Yaskawa INFORM job: SMPL0-B1.JBI

/JOB
//NAME SMPL0-B1
///FOLDERNAME INNE
//POS
///NPOS 7,7,0,0,0,0
///TOOL 0
///POSTYPE PULSE
///PULSE
C00000=-15600,-38077,-45406,-15836,-36040,13556
C00001=-14419,-31953,-44456,-15790,-33342,13448
C00002=-14246,-29435,-43033,-15820,-32912,13443
C00003=-13134,-13894,-31875,-15218,-31619,13038
C00004=-11137,-6393,-26538,-13470,-30721,11945
C00005=-12696,-9506,-25886,-14225,-32926,12476
C00006=-15600,-38077,-45406,-15836,-36040,13556
BC00000=-1640,-38077,-45406
BC00001=-1640,-38077,-45406
BC00002=-1640,-38077,-45406
BC00003=-1640,-38077,-45406
BC00004=-1640,-38077,-45406
BC00005=-1640,-38077,-45406
BC00006=-1640,-38077,-45406
//INST
///DATE 2023/10/04 15:13
///ATTR SC,RW
///GROUP1 RB1,BS1
///LVARS 0,0,0,0,0,0,0,0
NOP
SFTOF
'-- TL mode [B000]-------------
'- 0:NO TRACKING, 1:TRACKING --
'------------------------------
SET B000 1
MOVJ C00000 BC00000 VJ=25.00
MOVL C00001 BC00001 V=166.7
MACRO1 MJ#(5) ARGFB000 ARGF40 ARGF100 ARGFC00002 ARGFBC00002 ARGF7
'arcon
MOVL C00003 BC00003 V=16.7
MACRO1 MJ#(9) ARGFB000 ARGF40
MOVL C00004 BC00004 V=16.7
'arcof
MACRO1 MJ#(3) ARGFB000
MOVL C00005 BC00005 V=166.7
MOVJ C00006 BC00006 VJ=25.00
END
